Staubli VAL3: HRAS_trial.dtx

dio dDio_bk = {link=BasicIO-1\%Q4}
dio dDio_f1_fit = {link=BasicIO-1\%Q3}
dio dDio_f1_secure = {link=BasicIO-1\%Q5}
dio dDio_f2_secure = {link=BasicIO-1\%Q5}
dio dDio_f3_secure = {link=BasicIO-1\%Q5}
dio dDio_t1_cy = {link=valve2}
dio dDio_t1_vb = {link=BasicIO-1\%Q1}
dio dDio_t1_vg
dio dDio_t1_vs = {link=fIn0}
dio dDio_t2_cy = {link=valve1}
dio dDio_t3_cy
dio dDio_t3_vb
dio dDio_t3_vg
dio dDio_t3_vs = {link=fIn0}
frame back_secure = {x=115.58673, y=51.100364, z=20, fatherId=fFrame_plate_2[0]}
frame f1 = {x=122.11, y=150.29, z=10, fatherId=fFrame_plate_1[0]}
frame f2 = {x=-27.94, y=157.28, z=10, fatherId=fFrame_plate_1[0]}
frame f3 = {x=76.91, y=29, z=10, fatherId=fFrame_plate_1[0]}
frame fFrame_bt = {x=20, y=51, z=5.05, fatherId=fFrame_plate_2[0]}
frame fFrame_fixture = {x=215, y=110.7, z=20.45, fatherId=fFrame_plate_2[0]}
frame fFrame_local = {rz=-45, fatherId=fFrame_ofs[0]}
frame fFrame_offset = {z=2.5, fatherId=fFrame_fixture[0]}
frame fFrame_ofs = {x=64, y=165, fatherId=fFrame_bt[0]}
frame fFrame_plate_1 = {x=-25.13, y=543.53, rz=179.999999, fatherId=fFrame_reverse[0]}
frame fFrame_plate_2 = {x=256.560574, y=565.662705, rz=-126.583221, fatherId=fFrame_reverse[0]}
frame fFrame_reverse = {z=-176.5, fatherId=world[0]}
frame fixture = {x=-479.290297, y=224.508367, z=-148, rz=-90.00005, fatherId=fFrame_reverse[0]}
frame frame_bk = {x=19, y=9.2, fatherId=back_secure[0]}
frame shelf = {x=-472.219676, y=345.637635, z=-165, rz=-90, fatherId=fFrame_reverse[0]}
mdesc mNomSpeed
mdesc mSlowSpeed = {accel=50, vel=10, decel=50}
num nNum_apporach_h = 10
num nNum_blow_delay = 1
num nNum_blow_h = 0.5
num nNum_cy_delay = 0.5
num nNum_press = 4
num nNum_safe_h = 100
pointRx f1pick = {x=43.79, y=-7, z=0.5, rz=-180, fatherId=shelf[0]}
pointRx f1picksafe = {x=43.79, y=-7, z=20, rz=-180, fatherId=shelf[0]}
pointRx f1place = {x=20, y=-19.98, rz=-180, fatherId=fixture[0]}
pointRx f1placesafe = {x=20, y=-19.98, z=20, rz=180, fatherId=fixture[0]}
pointRx f2pick = {x=29.79, y=-6.4, z=0.5, rx=-180, rz=180, fatherId=shelf[0]}
pointRx f2picksafe = {x=29.79, y=-6.4, z=20, rx=-180, rz=179, fatherId=shelf[0]}
pointRx f2place = {x=20, y=-16.82, rz=-180, fatherId=fixture[0]}
pointRx f2placesafe = {x=20, y=-16.82, z=20, rz=180, fatherId=fixture[0]}
pointRx f3pick = {x=7.79, y=-6.75, z=0.5, rx=-180, wrist=wpositive, fatherId=shelf[0]}
pointRx f3picksafe = {x=7.790741, y=-6.500263, z=50, rx=-179.999806, ry=-0.000248, rz=-2.000096, fatherId=shelf[0]}
pointRx f3place = {x=20, y=-16.62, z=3.8, fatherId=fixture[0]}
pointRx f3placesafe = {x=20.000011, y=-16.619972, z=20, ry=0.000116, rz=0.000003, fatherId=fixture[0]}
pointRx ori = {rx=180, fatherId=fFrame_plate_1[0]}
pointRx orig = {rx=180, rz=45, fatherId=fFrame_plate_2[0]}
pointRx origin = {rz=-180, fatherId=fixture[0]}
pointRx pPointRx_bt_lb = {rx=-180, ry=0, rz=90, fatherId=fFrame_local[0]}
pointRx pPointRx_bt_pos = {rx=-0.000015, ry=-179.99988, rz=-90, fatherId=fFrame_offset[0]}
pointRx pPointRx_f1_bk = {y=-3, rx=180, ry=0, rz=-2, fatherId=frame_bk[0]}
pointRx pPointRx_f1_lb = {z=-2, rx=180, fatherId=f1[0]}
pointRx pPointRx_f1_pos = {x=0.2, y=-2.5, z=2.5, rx=180, fatherId=fFrame_offset[0]}
pointRx pPointRx_f2_bk = {x=-0.12, y=-0.4, rx=180, ry=0, rz=-1, fatherId=frame_bk[0]}
pointRx pPointRx_f2_lb = {z=-0.5, rx=180, fatherId=f2[0]}
pointRx pPointRx_f3_bk = {rx=180, rz=90, fatherId=frame_bk[0]}
pointRx pPointRx_f3_lb = {z=-2, rx=180, fatherId=f3[0]}
pointRx pPointRx_f3_pos = {y=-0.05, rx=180, ry=0, rz=87.75, fatherId=fFrame_offset[0]}
pointRx ref = {x=-188.838954, y=475.816737, z=20, rx=180, rz=180, fatherId=fFrame_reverse[0]}
screen sScreen_menu
screen sScreen_ppShelf
tool ca = {z=30, fatherId=flange[0], ioLink=valve1}
tool t1 = {y=47, z=94, fatherId=ca[0], ioLink=BasicIO-1\%Q0, ioOpen=1, ioClose=1}
tool t2 = {x=-47, z=94, fatherId=ca[0], ioLink=BasicIO-1\%Q1, ioOpen=0.5, ioClose=1}
tool t3 = {x=47, z=89.5, fatherId=ca[0], ioLink=BasicIO-1\%Q2, ioOpen=0.5, ioClose=1}
